Staubli VAL3: sendFbkMsg.pgx

public program sendFbkMsg(RobotStatus& x_rRobotStatus, FlagStatus& x_fRosStatus)
begin

  //This program is used for sending the robot feedback data to the host ROS controller and
  //ensure the data sent correct.

  while true
    //call the send data function
    call sendData(soTcpIpFbk,nSendData,x_rRobotStatus,x_fRosStatus)

    //Froce an end to the current task and enter the next sequence loop.
    delay(0.0)

  endWhile



end
